// TIA Portal V20 export
// export: Created 2026-07-14T21:19:13.6271096Z, ExportSetting WithDefaults, DisplayName Totally Integrated Automation Portal, DisplayVersion V20 Update 5, DisplayName TIA Portal Openness, DisplayVersion V20 Update 4, DisplayName TIA Portal Version Control Interface, DisplayVersion V20 Update 5, DisplayName SINAMICS Startdrive Advanced, DisplayVersion V20, DisplayName SINAMICS DCC, DisplayVersion V20, DisplayName SINAMICS Startdrive G130, G150, S120, S150, SINAMICS MV, G220, S200, S210, DisplayVersion V20, DisplayName SINAMICS Startdrive G110M, G120, G120C, G120D, G120P, G115D, DisplayVersion V20, DisplayName STEP 7 Professional, DisplayVersion V20 Update 5, DisplayName STEP 7 Safety, DisplayVersion V20 Update 2, DisplayName WinCC Basic/Comfort/Advanced, DisplayVersion V20 Update 5, DisplayName WinCC Unified, DisplayVersion V20 Update 5
FUNCTION "PerimeterSafetyAlarms" : Void   // FC18, LAD
TITLE = Perimeter Safety Alarms
{ S7_Optimized_Access := 'TRUE' }
VERSION : 0.1
// Packs perimeter-related safety and fire-damper field alarms into AlarmWords.AlarmWord1 for HMI display.
// stored: AutoNumber true, IsIECCheckEnabled false, SetENOAutomatically false, UDAEnableTagReadback false
BEGIN

REGION Network 1: Perimeter Safety Alarm Bit Mapping
   // Bits 0-4 are negated because SafetyZone1-3/SafetyGate1 read true when the circuit is intact, so a break reads false and NOT is what raises the alarm. Bits 5-7 are not negated: PullCord1/FireDamper1/FireDamper2 already report true-when-triggered from the field device. Bit 0 summarizes bits 1-3 (any zone breach) so the HMI can show one perimeter-alarm indicator without decoding the individual bits.
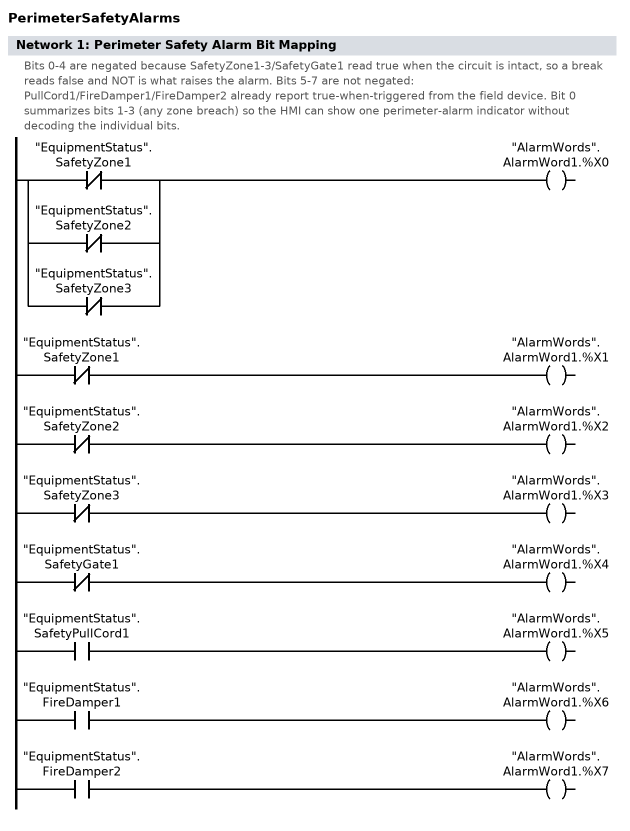
   RUNG wire#powerrail
      I_Contact( "EquipmentStatus".SafetyZone1 )
      wire#w1
      Coil( "AlarmWords".AlarmWord1.%X0 )
   END_RUNG
   RUNG wire#powerrail
      I_Contact( "EquipmentStatus".SafetyZone2 )
   END_RUNG wire#w1
   RUNG wire#powerrail
      I_Contact( "EquipmentStatus".SafetyZone3 )
   END_RUNG wire#w1
   RUNG wire#powerrail
      I_Contact( "EquipmentStatus".SafetyZone1 )
      Coil( "AlarmWords".AlarmWord1.%X1 )
   END_RUNG
   RUNG wire#powerrail
      I_Contact( "EquipmentStatus".SafetyZone2 )
      Coil( "AlarmWords".AlarmWord1.%X2 )
   END_RUNG
   RUNG wire#powerrail
      I_Contact( "EquipmentStatus".SafetyZone3 )
      Coil( "AlarmWords".AlarmWord1.%X3 )
   END_RUNG
   RUNG wire#powerrail
      I_Contact( "EquipmentStatus".SafetyGate1 )
      Coil( "AlarmWords".AlarmWord1.%X4 )
   END_RUNG
   RUNG wire#powerrail
      Contact( "EquipmentStatus".SafetyPullCord1 )
      Coil( "AlarmWords".AlarmWord1.%X5 )
   END_RUNG
   RUNG wire#powerrail
      Contact( "EquipmentStatus".FireDamper1 )
      Coil( "AlarmWords".AlarmWord1.%X6 )
   END_RUNG
   RUNG wire#powerrail
      Contact( "EquipmentStatus".FireDamper2 )
      Coil( "AlarmWords".AlarmWord1.%X7 )
   END_RUNG
   // the same network as SCL:
   "AlarmWords".AlarmWord1.%X0 := NOT "EquipmentStatus".SafetyZone1 OR NOT "EquipmentStatus".SafetyZone2 OR NOT "EquipmentStatus".SafetyZone3;
   "AlarmWords".AlarmWord1.%X1 := NOT "EquipmentStatus".SafetyZone1;
   "AlarmWords".AlarmWord1.%X2 := NOT "EquipmentStatus".SafetyZone2;
   "AlarmWords".AlarmWord1.%X3 := NOT "EquipmentStatus".SafetyZone3;
   "AlarmWords".AlarmWord1.%X4 := NOT "EquipmentStatus".SafetyGate1;
   "AlarmWords".AlarmWord1.%X5 := "EquipmentStatus".SafetyPullCord1;
   "AlarmWords".AlarmWord1.%X6 := "EquipmentStatus".FireDamper1;
   "AlarmWords".AlarmWord1.%X7 := "EquipmentStatus".FireDamper2;
END_REGION
END_FUNCTION
